DATA_BLOCK "DB_Int_Programming"
TITLE =%version: 0.04 % CN: 20
//This version  %created_by: nlhdl %
//              %date_created: maandag 6 juli 2015 10:22:58 %
//              %release: VI_CONV/RA_Dev_Oakham %
//
//Modification History:                                   By:    Date:     Rev:
//----------------------------------------------------  -------  --------  -----
//7324: ECS-P General from the RD to RA for platform    nlHdL    06-07-15   0.04
//15797: Keyword release added                          nlwwij   26-09-13   0.04
//CR8000 Remove example code                            nlple     28-11-11  0.03
//CR7631 Insert key word for code generator             nlple     06-10-11  0.02
//Initial version                                       nlMvK     20-10-10  0.01
//
FAMILY : General
VERSION : 0.0


  STRUCT
   Insert : INT ;	// Insertion point for the S7 Code Generator
  END_STRUCT ;
BEGIN
   Insert := 0;
END_DATA_BLOCK

